// Mitsubishi GX Works2 project: test   PLC: Q03UDV

PROGRAM MAIN
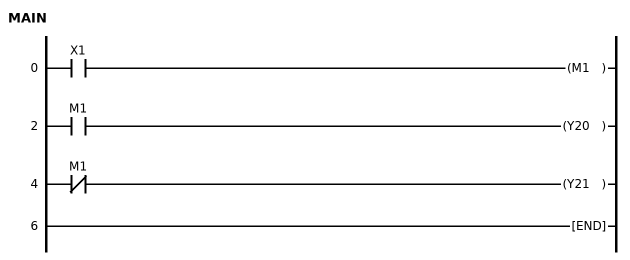
0     LD      X1
      OUT     M1
2     LD      M1
      OUT     Y20
4     LDI     M1
      OUT     Y21
6     END
END_PROGRAM
